FUNCTION_BLOCK POU
VAR_INPUT
END_VAR
VAR_OUTPUT
END_VAR
VAR
	a , b, c : INT := 5;
	d : INT ;
END_VAR

d := a+b+c+d;

END_FUNCTION_BLOCK

(* stored: Version 1.1.0.1, ProductVersion 3.1.4024.9
   POU POU: Id {06e6837e-abdc-4596-b423-197af08c097a}, SpecialFunc None *)
